// TIA Portal V17 export
// export: Created 2022-07-20T06:59:47.9831804Z, ExportSetting WithDefaults, DisplayName Totally Integrated Automation Portal, DisplayVersion V17, DisplayName TIA Portal Openness, DisplayVersion V17, DisplayName TIA Portal Version Control Interface, DisplayVersion V17, DisplayName SINAMICS Startdrive Advanced, DisplayVersion V17, DisplayName SINAMICS Startdrive G130, G150, S120, S150, SINAMICS MV, S210, DisplayVersion V17, DisplayName SINAMICS Startdrive G110M, G120, G120C, G120D, G120P, G115D, DisplayVersion V17, DisplayName STEP 7 Professional, DisplayVersion V17, DisplayName STEP 7 Safety, DisplayVersion V17, DisplayName WinCC Advanced, DisplayVersion V17
FUNCTION_BLOCK "FB10190_PaperJam"   // FB10190, LAD
TITLE = FB10190_PaperJam
{ S7_Optimized_Access := 'TRUE' }
AUTHOR : Anirouddh
FAMILY : 1019_TRANSPORT
VERSION : 1.0
// Release note : 
// 1.0 - Feature developped
// stored: AutoNumber false, IsIECCheckEnabled false, IsRetainMemResEnabled false, MemoryReserve 100, SetENOAutomatically false, UDAEnableTagReadback false
   VAR_INPUT
      FirstSheetSensor : Bool;
      SecondSheetSensor : Bool;
      SheetSize : Real;   // mm
      TransportSpeed : Real;   // mm/s
      Margin : Real;   // 0-100%
      DistanceBetweenSheetSensors : Real;
      Reset : Bool;
   END_VAR
   VAR_OUTPUT
      PaperJamDetected : Bool;
   END_VAR
   VAR
      i : SInt;
      R_TRIG_FirstSensorSignal { S7_SetPoint := 'True'} : R_TRIG;
      F_TRIG_FirstSensorSignal { S7_SetPoint := 'True'} : F_TRIG;
      R_TRIG_SecondSensorSignal { S7_SetPoint := 'True'} : R_TRIG;
      F_TRIG_SecondSensorSignal { S7_SetPoint := 'True'} : F_TRIG;
      SheetsRegistration_RTRIG_S1 : Array[0..49] of Bool;
      SheetsRegistration_FTRIG_S1 : Array[0..49] of Bool;
      SheetsRegistration_RTRIG_S2 : Array[0..49] of Bool;
      SheetsRegistration_FTRIG_S2 : Array[0..49] of Bool;
      TON_SheetsRegistration_UnderFirstSensor : Array[0..49] of TON_TIME;
      TON_SheetsRegistration_UnderSecondSensor : Array[0..49] of TON_TIME;
      TON_SheetsRegistration_BetweenSensors { S7_SetPoint := 'True'} : Array[0..49] of TON_TIME;
   END_VAR
BEGIN

REGION Network 1 (SCL): First Scan
   IF "FirstScan" THEN
       FOR #i:= 0 TO 49 DO
           #SheetsRegistration_RTRIG_S1[#i] := FALSE;
           #SheetsRegistration_FTRIG_S1[#i] := FALSE;
           #SheetsRegistration_RTRIG_S2[#i] := FALSE;
           #SheetsRegistration_FTRIG_S2[#i] := FALSE;
           RESET_TIMER(#TON_SheetsRegistration_UnderFirstSensor[#i]);
           RESET_TIMER(#TON_SheetsRegistration_UnderSecondSensor[#i]);
           RESET_TIMER(#TON_SheetsRegistration_BetweenSensors[#i]);
       END_FOR;
   END_IF;
END_REGION

REGION Network 2 (SCL): Edge Signals & Timers
   REGION EDGE SIGNALS
       #R_TRIG_FirstSensorSignal(CLK := #FirstSheetSensor);
       #F_TRIG_FirstSensorSignal(CLK := #FirstSheetSensor);
       #R_TRIG_SecondSensorSignal(CLK := #SecondSheetSensor);
       #F_TRIG_SecondSensorSignal(CLK := #SecondSheetSensor);
   END_REGION

   REGION TIMERS
       FOR #i := 0 TO 49 DO
           #TON_SheetsRegistration_UnderFirstSensor[#i](IN := #SheetsRegistration_RTRIG_S1[#i] AND NOT (#SheetsRegistration_FTRIG_S1[#i]),
                                                         PT := DINT_TO_TIME(REAL_TO_DINT((1 + (#Margin / 100.0)) * (#SheetSize / #TransportSpeed)) * 1000));
           #TON_SheetsRegistration_UnderSecondSensor[#i](IN := #SheetsRegistration_RTRIG_S2[#i] AND NOT (#SheetsRegistration_FTRIG_S2[#i]),
                                                          PT := DINT_TO_TIME(REAL_TO_DINT((1 + (#Margin / 100.0)) * (#SheetSize / #TransportSpeed)) * 1000));
           #TON_SheetsRegistration_BetweenSensors[#i](IN := #SheetsRegistration_RTRIG_S1[#i] AND NOT (#SheetsRegistration_FTRIG_S2[#i]),
                                                       PT := DINT_TO_TIME(REAL_TO_DINT((1 + (#Margin / 100.0)) * ((#DistanceBetweenSheetSensors + #SheetSize) / #TransportSpeed) * 1000)));
       END_FOR;
   END_REGION
END_REGION

REGION Network 3 (SCL): Edges Detection Management
   //Detect to Rising Edge of the first sensor
   IF #R_TRIG_FirstSensorSignal.Q THEN
       FOR #i := 0 TO 49 DO
           IF NOT (#SheetsRegistration_RTRIG_S1[#i]) THEN
               #SheetsRegistration_RTRIG_S1[#i] := TRUE;
               EXIT;
           END_IF;
       END_FOR;
   END_IF;

   //Detect the falling edge of the first sensor
   IF #F_TRIG_FirstSensorSignal.Q THEN
       FOR #i := 0 TO 49 DO
           IF NOT (#SheetsRegistration_FTRIG_S1[#i]) THEN
               #SheetsRegistration_FTRIG_S1[#i] := TRUE;
               EXIT;
           END_IF;
       END_FOR;
   END_IF;

   //Detect the rising edge OF the second sensor
   IF #R_TRIG_SecondSensorSignal.Q THEN
       FOR #i := 0 TO 49 DO
           IF NOT (#SheetsRegistration_RTRIG_S2[#i]) THEN
               #SheetsRegistration_RTRIG_S2[#i] := TRUE;
               EXIT;
           END_IF;
       END_FOR;
   END_IF;

   //Detect the falling edge of the second sensor
   IF #F_TRIG_SecondSensorSignal.Q THEN
       FOR #i := 0 TO 49 DO
           IF NOT (#SheetsRegistration_FTRIG_S2[#i]) THEN
               #SheetsRegistration_FTRIG_S2[#i] := TRUE;
               EXIT;
           END_IF;
       END_FOR;
   END_IF;
END_REGION

REGION Network 4 (SCL): Jam Management
   //Sensor Alone Jam Management
   FOR #i := 0 TO 49 DO
       //First Sensor Jam Management
       IF #TON_SheetsRegistration_UnderFirstSensor[#i].Q AND #SheetsRegistration_RTRIG_S1[#i] AND NOT (#SheetsRegistration_FTRIG_S1[#i]) THEN
           #PaperJamDetected := TRUE;
       END_IF;

       //Second Sensor Jam Management
       IF #TON_SheetsRegistration_UnderSecondSensor[#i].Q AND #SheetsRegistration_RTRIG_S2[#i] AND NOT (#SheetsRegistration_FTRIG_S2[#i]) THEN
           #PaperJamDetected := TRUE;
       END_IF;
   END_FOR;

   //Between Sensor Jam Management
   IF #TON_SheetsRegistration_BetweenSensors[0].Q THEN
       IF NOT (#SheetsRegistration_RTRIG_S1[0]) OR NOT (#SheetsRegistration_FTRIG_S1[0]) OR NOT (#SheetsRegistration_RTRIG_S2[0]) OR NOT (#SheetsRegistration_FTRIG_S2[0]) THEN
           #PaperJamDetected := TRUE;
       ELSE
           #SheetsRegistration_RTRIG_S1[0] := FALSE;
           #SheetsRegistration_FTRIG_S1[0] := FALSE;
           #SheetsRegistration_RTRIG_S2[0] := FALSE;
           #SheetsRegistration_FTRIG_S2[0] := FALSE;
       END_IF;
       FOR #i := 1 TO 49 DO
           #SheetsRegistration_RTRIG_S1[#i - 1] := #SheetsRegistration_RTRIG_S1[#i];
           #SheetsRegistration_FTRIG_S1[#i - 1] := #SheetsRegistration_FTRIG_S1[#i];
           #SheetsRegistration_RTRIG_S2[#i - 1] := #SheetsRegistration_RTRIG_S2[#i];
           #SheetsRegistration_FTRIG_S2[#i - 1] := #SheetsRegistration_FTRIG_S2[#i];
       END_FOR;
   END_IF;
END_REGION

REGION Network 5 (SCL): Reset Jam
   IF #Reset AND NOT (#FirstSheetSensor) AND NOT (#SecondSheetSensor) THEN
       #PaperJamDetected := FALSE;
       FOR #i := 0 TO 49 DO
           #SheetsRegistration_RTRIG_S1[#i] := FALSE;
           #SheetsRegistration_FTRIG_S1[#i] := FALSE;
           #SheetsRegistration_RTRIG_S2[#i] := FALSE;
           #SheetsRegistration_FTRIG_S2[#i] := FALSE;
           RESET_TIMER(#TON_SheetsRegistration_BetweenSensors[#i]);
       END_FOR;
   END_IF;
END_REGION
END_FUNCTION_BLOCK
